(* PLC project int2real_scale, Dassault Systèmes ControlBuild 2024x *)
(* stored: creationDateTime 2023-10-03T11:13:31-01:00 *)

(* This module simulates a scaling of an integer into a real. Form of the scaling equation is y = k x . *)
FUNCTION_BLOCK equipment_library.int2real_scale
  VAR_INPUT
    inputValueD : DINT := 0;
    inputValueI : INT := 0;
  END_VAR
  VAR_OUTPUT
    outputValue : REAL := 0.0;
  END_VAR
  VAR CONSTANT
    coefficient : REAL := 1.0;
    offset : REAL := 0.0;
    selectDouble : BOOL := true;
  END_VAR
  VAR
    d_scale : BOOL := false;
    v_d_scale : REAL := 10.0;
  END_VAR


ACTION C_source_code:
/* ----------------------------------------------------------------	*/
/* Type : Model of Operative Behaviour					*/
/* Category :  Toolbox							*/
/* Author : Dassault Systemes						*/
/* Update date : June 2018						*/
/* ----------------------------------------------------------------	*/
/* This module simulates a scaling of an integer into a real	 	*/
/*	by multiplying it by a parameter coefficient.			*/
/* Form of the scaling equation is y = k x .				*/
/* ----------------------------------------------------------------	*/

if (d_scale)
	outputValue = v_d_scale;
else {
	if (selectDouble) outputValue = (inputValueD * coefficient) + offset;
	else outputValue = (inputValueI * coefficient) + offset ;
}
END_ACTION
END_FUNCTION_BLOCK
